// TIA Portal V17 export
// export: Created 2025-08-05T09:35:54.7845652Z, ExportSetting WithDefaults, DisplayName Totally Integrated Automation Portal, DisplayVersion V17, DisplayName TIA Portal Openness, DisplayVersion V17, DisplayName TIA Portal Version Control Interface, DisplayVersion V17, DisplayName SINAMICS Startdrive Advanced, DisplayVersion V17, DisplayName SINAMICS Startdrive G130, G150, S120, S150, SINAMICS MV, S210, DisplayVersion V17, DisplayName SINAMICS Startdrive G110M, G120, G120C, G120D, G120P, G115D, DisplayVersion V17, DisplayName STEP 7 Professional, DisplayVersion V17, DisplayName STEP 7 Safety, DisplayVersion V17, DisplayName WinCC Advanced, DisplayVersion V17
FUNCTION_BLOCK "GraphEvaluation"   // FB38, LAD
TITLE = S7 graph evaluation / S7-Graph Auswertung
{ S7_Optimized_Access := 'TRUE' }
AUTHOR : Grob
FAMILY : Kernel_V2
VERSION : 1.4
// S7 graph evaluation / S7-Graph Auswertung
// stored: AutoNumber true, IsIECCheckEnabled true, IsRetainMemResEnabled false, MemoryReserve 100, SetENOAutomatically true, UDAEnableTagReadback false
   VAR_INPUT
      rtData { ExternalAccessible := 'False'; ExternalVisible := 'False'; ExternalWritable := 'False'} : G7_RTDataPlus_V6;   // Graph RT_DATA
      timeOutTime { ExternalAccessible := 'False'; ExternalVisible := 'False'; ExternalWritable := 'False'} : Time := T#5m;   // Timeout Zeit / Timeout time
   END_VAR
   VAR_OUTPUT
      timeOut { ExternalAccessible := 'False'; ExternalVisible := 'False'; ExternalWritable := 'False'} : Bool;   // Timeout Fehler / Timeout error
   END_VAR
   VAR_IN_OUT
      funcGrp : "typeCaCgFg";   // Funktionsgruppe / Function Group
      fgControlGeneral : "typeFgControlGeneral";   // Funktionsgruppe Allgemeine Steuerschnittstelle / General control interface function group
   END_VAR
   VAR
      statErrorTimeOut { ExternalAccessible := 'False'; ExternalVisible := 'False'; ExternalWritable := 'False'} : Bool;   // ProDiag-Störung: Timeout / ProDiag fault: Timeout
      statCount { ExternalAccessible := 'False'; ExternalVisible := 'False'; ExternalWritable := 'False'} : USInt;   // Zähler / Counter
      statFgName { ExternalAccessible := 'False'; ExternalVisible := 'False'; ExternalWritable := 'False'} : WString["GRP_JOB_NAME_SIZE"];   // ProDiag Begleitwert: Name der FG / ProDiag associated value: Name of the FG
      statGraphStepNumber { ExternalAccessible := 'False'; ExternalVisible := 'False'; ExternalWritable := 'False'} : Int;   // ProDiag Begleitwert: Schrittnummer / ProDiag associated value: step number
      statLastStepNumber { ExternalAccessible := 'False'; ExternalVisible := 'False'; ExternalWritable := 'False'} : Int;   // Letzte Schrittnummer gespeichert / Last step number saved
      instTimerTimeOut { ExternalAccessible := 'False'; ExternalVisible := 'False'; ExternalWritable := 'False'} : TON_TIME;   // Timer Timeout / Timer for timeout
   END_VAR
BEGIN

REGION Network 1 (SCL): Version
   //===============================================================================================================================
   // GROB-WERKE GmbH & Co. KG
   // (c)Copyright 2022 All Rights Reserved
   //
   // Reproduction, replication, modification, distribution, communication to the public and making the work available to the public
   // or others as well as other exploitation of the software and, if applicable, the medium containing the software without express
   // authorization is prohibited. Offenders will be held liable for the payment of damages. All rights reserved with regard to the
   // protection of intellectual property
   // ------------------------------------------------------------------------------------------------------------------------------
   //     Library:       Kernel V2
   //     Tested with:   PLCSIM
   //     Engineering:   TIA Portal V17
   //     Restrictions:  ---
   //     Requirements:  ---
   REGION Functionality
       //                This function block has to be  called in the permanent post-instructions
       //
       //                It evaluates information of the graph and writes informations to the function group
       //                control interface (typeFgControlGeneral in Fg*General-DB)
       //                Further it triggers stop to the function group in single step mode after finishing a sequence step
       //
       //                Handles the general graph step time out
   END_REGION
   // ------------------------------------------------------------------------------------------------------------------------------
   // Change log table: 
   //     Version    Date      Expert in charge    Changes applied 
   //     -------|------------|-----------------|-----------------------------------------------------------------------------------
   //     00.00    24.05.2022  Dorn, F.            Migrated from TST V1.4, block version 01.00
   //     01.00    24.05.2022  Dorn, F.            First released version
   //     01.01    02.08.2022  Dorn, F.            Reset functiongroup after graph reinitialization
   //     01.02    21.11.2022  Dorn, F.            Fixed graph time out. (caused 2 alarms)
   //     01.03    18.02.2023  Dorn, F.            Implemented new internal signals in typeFgControlGeneral 
   //                                                  (start delays for GraphControl-funciton)
   //     01.04    18.12.2023  Dorn, F.            Implemented signals for stop selected by...
   //===============================================================================================================================
END_REGION

REGION Network 3: *************** General *************** / *************** Allgemein ***************
END_REGION

REGION Network 4: Graph fault sent to group / Graph Störung an Gruppe übertragen
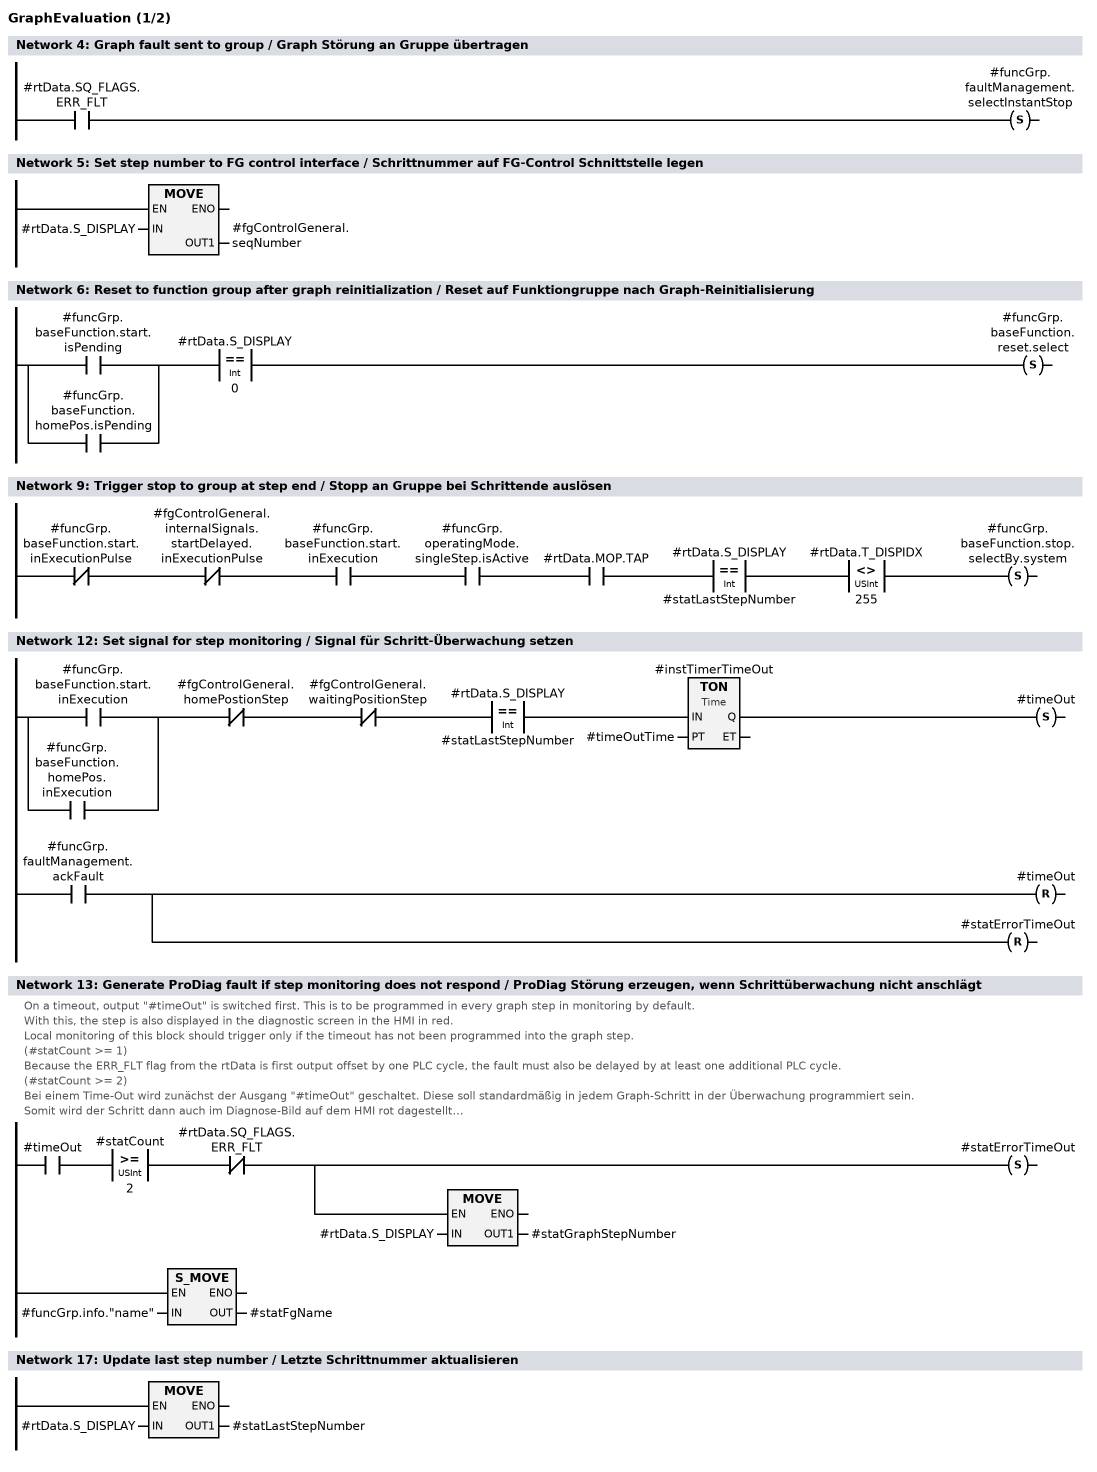
   RUNG wire#powerrail
      Contact( #rtData.SQ_FLAGS.ERR_FLT )
      S_Coil( #funcGrp.faultManagement.selectInstantStop )
   END_RUNG
   // the same network as SCL:
   IF #rtData.SQ_FLAGS.ERR_FLT THEN #funcGrp.faultManagement.selectInstantStop := TRUE; END_IF;
END_REGION

REGION Network 5: Set step number to FG control interface / Schrittnummer auf FG-Control Schnittstelle legen
   RUNG wire#powerrail
      Move(in := #rtData.S_DISPLAY, out1 => #fgControlGeneral.seqNumber)
   END_RUNG
   // the same network as SCL:
   #fgControlGeneral.seqNumber := #rtData.S_DISPLAY;
END_REGION

REGION Network 6: Reset to function group after graph reinitialization / Reset auf Funktiongruppe nach Graph-Reinitialisierung
   RUNG wire#powerrail
      Contact( #funcGrp.baseFunction.start.isPending )
      wire#w1
      { S7_Templates := "SrcType := Int" } EQ_Contact(in1 := #rtData.S_DISPLAY, in2 := 0)
      S_Coil( #funcGrp.baseFunction.reset.select )
   END_RUNG
   RUNG wire#powerrail
      Contact( #funcGrp.baseFunction.homePos.isPending )
   END_RUNG wire#w1
   // the same network as SCL:
   IF (#funcGrp.baseFunction.start.isPending OR #funcGrp.baseFunction.homePos.isPending) AND (#rtData.S_DISPLAY = 0) THEN
       #funcGrp.baseFunction.reset.select := TRUE;
   END_IF;
END_REGION

REGION Network 8: *************** Single-step (TAP) *************** / *************** Einzelschritt (TAP) ***************
END_REGION

REGION Network 9: Trigger stop to group at step end / Stopp an Gruppe bei Schrittende auslösen
   RUNG wire#powerrail
      I_Contact( #funcGrp.baseFunction.start.inExecutionPulse )
      I_Contact( #fgControlGeneral.internalSignals.startDelayed.inExecutionPulse )
      Contact( #funcGrp.baseFunction.start.inExecution )
      Contact( #funcGrp.operatingMode.singleStep.isActive )
      Contact( #rtData.MOP.TAP )
      { S7_Templates := "SrcType := Int" } EQ_Contact(in1 := #rtData.S_DISPLAY, in2 := #statLastStepNumber)
      { S7_Templates := "SrcType := USInt" } NE_Contact(in1 := #rtData.T_DISPIDX, in2 := 255)
      S_Coil( #funcGrp.baseFunction.stop.selectBy.system )
   END_RUNG
   // the same network as SCL:
   IF NOT #funcGrp.baseFunction.start.inExecutionPulse AND NOT #fgControlGeneral.internalSignals.startDelayed.inExecutionPulse AND #funcGrp.baseFunction.start.inExecution AND #funcGrp.operatingMode.singleStep.isActive AND #rtData.MOP.TAP AND (#rtData.S_DISPLAY = #statLastStepNumber) AND (#rtData.T_DISPIDX <> 255) THEN
       #funcGrp.baseFunction.stop.selectBy.system := TRUE;
   END_IF;
END_REGION

REGION Network 11: *************** Timeout monitoring *************** / *************** Timeout Überwachung ***************
END_REGION

REGION Network 12: Set signal for step monitoring / Signal für Schritt-Überwachung setzen
   RUNG wire#powerrail
      Contact( #funcGrp.baseFunction.start.inExecution )
      wire#w1
      I_Contact( #fgControlGeneral.homePostionStep )
      I_Contact( #fgControlGeneral.waitingPositionStep )
      { S7_Templates := "SrcType := Int" } EQ_Contact(in1 := #rtData.S_DISPLAY, in2 := #statLastStepNumber)
      { S7_Templates := "time_type := Time" } #instTimerTimeOut.TON(pt := #timeOutTime, et =>)
      S_Coil( #timeOut )
   END_RUNG
   RUNG wire#powerrail
      Contact( #funcGrp.baseFunction.homePos.inExecution )
   END_RUNG wire#w1
   RUNG wire#powerrail
      Contact( #funcGrp.faultManagement.ackFault )
      wire#w2
      R_Coil( #timeOut )
   END_RUNG
   RUNG wire#w2
      R_Coil( #statErrorTimeOut )
   END_RUNG
   // the same network as SCL:
   #instTimerTimeOut(IN := (#funcGrp.baseFunction.start.inExecution OR #funcGrp.baseFunction.homePos.inExecution) AND NOT #fgControlGeneral.homePostionStep AND NOT #fgControlGeneral.waitingPositionStep AND (#rtData.S_DISPLAY = #statLastStepNumber),   // TON
                     PT := #timeOutTime);
   IF #instTimerTimeOut.Q THEN #timeOut := TRUE; END_IF;
   IF #funcGrp.faultManagement.ackFault THEN
       #timeOut := FALSE;
       #statErrorTimeOut := FALSE;
   END_IF;
END_REGION

REGION Network 13: Generate ProDiag fault if step monitoring does not respond / ProDiag Störung erzeugen, wenn Schrittüberwachung nicht anschlägt
   // On a timeout, output "#timeOut" is switched first. This is to be programmed in every graph step in monitoring by default.
   // With this, the step is also displayed in the diagnostic screen in the HMI in red.
   // Local monitoring of this block should trigger only if the timeout has not been programmed into the graph step.
   // (#statCount >= 1)
   // 
   // Because the ERR_FLT flag from the rtData is first output offset by one PLC cycle, the fault must also be delayed by at least one additional PLC cycle.
   // (#statCount >= 2)
   // Bei einem Time-Out wird zunächst der Ausgang "#timeOut" geschaltet. Diese soll standardmäßig in jedem Graph-Schritt in der Überwachung programmiert sein.
   // Somit wird der Schritt dann auch im Diagnose-Bild auf dem HMI rot dagestellt.
   // Nur, wenn der Time-Out im Graphschritt nicht programmeirt wurde, soll die lokale Überwachung von diesem Baustein auslösen.
   // (#statCount >= 1)
   // 
   // Da das Flag ERR_FLT vom den rtData erst um einen PLC-Zyklus versetzt ausgegeben wird, muss die Störung zusätzlich noch um mindestens einen PLC-Zyklus  verzögert werden.
   // (#statCount >= 2)
   RUNG wire#powerrail
      Contact( #timeOut )
      { S7_Templates := "SrcType := USInt" } GE_Contact(in1 := #statCount, in2 := 2)
      I_Contact( #rtData.SQ_FLAGS.ERR_FLT )
      wire#w1
      S_Coil( #statErrorTimeOut )
   END_RUNG
   RUNG wire#w1
      Move(in := #rtData.S_DISPLAY, out1 => #statGraphStepNumber)
   END_RUNG
   RUNG wire#powerrail
      S_Move(in := #funcGrp.info."name", out => #statFgName)
   END_RUNG
   // the same network as SCL:
   IF #timeOut AND (#statCount >= 2) AND NOT #rtData.SQ_FLAGS.ERR_FLT THEN
       #statErrorTimeOut := TRUE;
       #statGraphStepNumber := #rtData.S_DISPLAY;
   END_IF;
   #statFgName := #funcGrp.info."name";
END_REGION

REGION Network 14 (SCL): Counter for fault / Zähler für Störung
   IF #timeOut AND NOT (#rtData.SQ_FLAGS.ERR_FLT OR #statErrorTimeOut) THEN
       #statCount += 1;
   ELSIF NOT #timeOut THEN
       #statCount := 0;
   END_IF;
END_REGION

REGION Network 16: *************** Internal control signals *************** / *************** Interne Steuersignale ***************
END_REGION

REGION Network 17: Update last step number / Letzte Schrittnummer aktualisieren
   RUNG wire#powerrail
      Move(in := #rtData.S_DISPLAY, out1 => #statLastStepNumber)
   END_RUNG
   // the same network as SCL:
   #statLastStepNumber := #rtData.S_DISPLAY;
END_REGION

REGION Network 18: Delayed start signals for "GraphControl"-FC / Verzögerte Start-Signale für "GraphControl"-FC
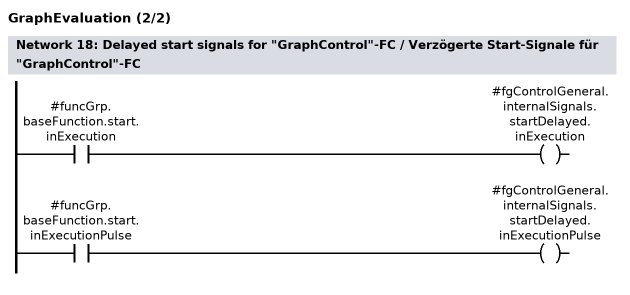
   RUNG wire#powerrail
      Contact( #funcGrp.baseFunction.start.inExecution )
      Coil( #fgControlGeneral.internalSignals.startDelayed.inExecution )
   END_RUNG
   RUNG wire#powerrail
      Contact( #funcGrp.baseFunction.start.inExecutionPulse )
      Coil( #fgControlGeneral.internalSignals.startDelayed.inExecutionPulse )
   END_RUNG
   // the same network as SCL:
   #fgControlGeneral.internalSignals.startDelayed.inExecution := #funcGrp.baseFunction.start.inExecution;
   #fgControlGeneral.internalSignals.startDelayed.inExecutionPulse := #funcGrp.baseFunction.start.inExecutionPulse;
END_REGION
END_FUNCTION_BLOCK
